TYPE ST_control_pannel :
STRUCT
	button_start		: BOOL;
	button_stop			: BOOL;
	button_reset		: BOOL;
	button_power		: BOOL;
	
	lamp_start			: BOOL;
	lamp_stop			: BOOL;
	lamp_reset			: BOOL;
	
END_STRUCT
END_TYPE

(* stored: Version 1.1.0.1, ProductVersion 3.1.4024.12
   DUT ST_control_pannel: Id {5868eef3-ea3b-4ed9-b395-503de9e035c4} *)
